PROGRAM N2Purge
VAR
	nSource: INT;
	nStartTimeInSeconds: UDINT ;
	nTime: UDINT;
	tempSecondsToAddWhilePause: DINT;
	SecondsToAddWhilePause: DINT;
	RemainingTime: UDINT;
	fb_FTRIG: R_TRIG;
	bStartCommand: BOOL;
	CLK: INT;
	Q: INT;
	b: BOOL;
	bN2PurgeBlockEnded: BOOL;
	fbSelection : FBSelection;
	

END_VAR

VAR_INPUT
	nCurrentBlock: INT;
	sSourceName: STRING;
END_VAR

fbSelection.TargetConverter(sTargetName:= sSourceName, TargetConverter_output => nSource); 

IF RecipeTags.Recipe.Blocks[nCurrentBlock].Properties.sStartTime = '' THEN
	RecipeTags.StaredTimeForRecipeBanner := MAIN.concatenatedHourMinuteString;
END_IF
IF (RecipeTags.bStartTimeEnable[nCurrentBlock]=FALSE) THEN
//	RecipeControl.StaredTimeForRecipeBanner := MAIN.concatenatedHourMinuteString;
	RecipeTags.Recipe.Blocks[nCurrentBlock].Properties.sStartTime:=MAIN.sConcatenatedHourMinuteString;
	nStartTimeInSeconds := STRING_TO_UDINT(MAIN.sCurrentSecond);
	RecipeTags.bStartTimeEnable[nCurrentBlock] :=  TRUE;
END_IF



IF RecipeTags.Recipe.Blocks[nCurrentBlock].Properties.sIntervalType = 'S' THEN
	nTime := DINT_TO_UDINT(RecipeTags.Recipe.Blocks[nCurrentBlock].Properties.nInterval);
ELSIF RecipeTags.Recipe.Blocks[nCurrentBlock].Properties.sIntervalType = 'M' THEN
	nTime := DINT_TO_UDINT(RecipeTags.Recipe.Blocks[nCurrentBlock].Properties.nInterval * 60);
ELSIF RecipeTags.Recipe.Blocks[nCurrentBlock].Properties.sIntervalType = 'H' THEN
	nTime := DINT_TO_UDINT(RecipeTags.Recipe.Blocks[nCurrentBlock].Properties.nInterval * 3600);
END_IF



IF RecipeTags.enWaitPause[nCurrentBlock] THEN
	tempSecondsToAddWhilePause := tempSecondsToAddWhilePause + 1;
	SecondsToAddWhilePause := tempSecondsToAddWhilePause; 
ELSE
	tempSecondsToAddWhilePause := 0;
	SecondsToAddWhilePause :=0;

END_IF

IF NOT(RecipeTags.bPauseRecipe) THEN
		RecipeTags.enWaitPause[nCurrentBlock] := FALSE;
		RecipeTags.bBlockStart[nCurrentBlock] := TRUE;
		RemainingTime := nTime- nStartTimeInSeconds-STRING_TO_UDINT(MAIN.sCurrentSecond);
ELSE
		RecipeTags.bBlockStart[nCurrentBlock] := FALSE;
		RecipeTags.enWaitPause[nCurrentBlock] := TRUE;
END_IF


IF  (nTime + nStartTimeInSeconds + DINT_TO_UDINT(TRUNC(SecondsToAddWhilePause/100))) <= (STRING_TO_UDINT(MAIN.sCurrentSecond)) THEN
	RecipeTags.Recipe.Blocks[nCurrentBlock].Properties.bStopCommand := TRUE;
	RecipeTags.Recipe.Blocks[nCurrentBlock].Properties.sEndTime:=MAIN.sConcatenatedHourMinuteString;
	RecipeTags.bBlockStart[nCurrentBlock] := FALSE;
	RecipeTags.bBlockEnd[nCurrentBlock] := TRUE;
ELSE
	RecipeTags.bBlockEnd[nCurrentBlock] := FALSE;

END_IF

IF RecipeTags.bBlockStart[nCurrentBlock] THEN
	IF nSource<9 THEN
		IO.Vessels[nSource].Valves[1].bStart := TRUE;
	END_IF
	IF nSource>=9 AND nSource<=11 THEN
		IO.Reactors[nSource-9].Valves[1].bStart := TRUE;
	END_IF
ELSE
	IF nSource<9 THEN
		IO.Vessels[nSource].Valves[1].bStart := FALSE;
	END_IF
	IF nSource>=9 AND nSource<=11 THEN
		IO.Reactors[nSource-9].Valves[1].bStart := FALSE;
	end_if
END_IF

fb_FTRIG(CLK:=RecipeTags.bBlockEnd[nCurrentBlock], Q=> );
IF fb_FTRIG.Q AND RecipeTags.Recipe.Blocks[nCurrentBlock].Name = 'N2Purge' THEN
	RecipeTags.Recipe.Blocks[nCurrentBlock].Properties.sEndTime:=MAIN.sConcatenatedHourMinuteString;
	RecipeTags.Recipe.Blocks[nCurrentBlock].Properties.bStopCommand := TRUE;
	RecipeTags.bBlockEnd[nCurrentBlock] := FALSE;
	RecipeTags.bStartTimeEnable[nCurrentBlock] :=  FALSE;

END_IF

END_PROGRAM

(* stored: Version 1.1.0.1, ProductVersion 3.1.4024.5
   POU N2Purge: Id {c101128e-3ae6-46fa-b4e9-38bad4c7d592}, SpecialFunc None *)
